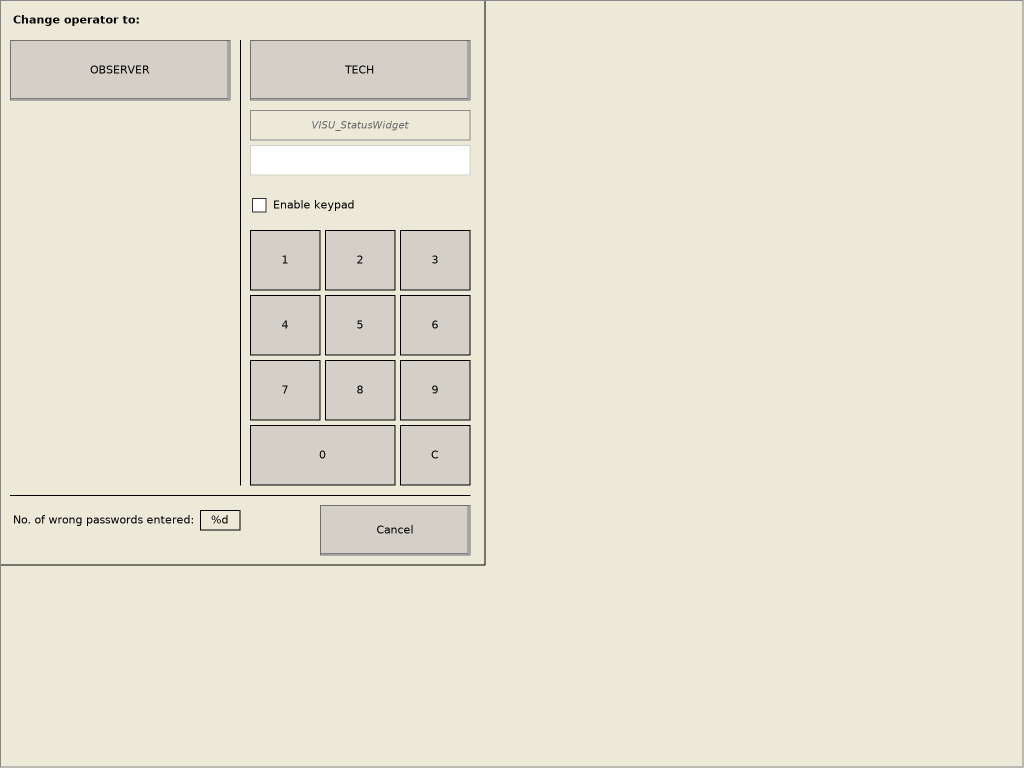
VISUALIZATION VISU_MTCSChangeOperatorDialog  // 1024x768
    Rectangle (0,0 485x565)
    Rectangle (250,230 70x60), "1", input disabled if: GLOBAL.gui.changeOperatorDialog.deactivate_keypad_keys
        OnMouseClick: execute { GLOBAL.gui.changeOperatorDialog.do_1 := TRUE; }
    Rectangle (325,230 70x60), "2", input disabled if: GLOBAL.gui.changeOperatorDialog.deactivate_keypad_keys
        OnMouseClick: execute { GLOBAL.gui.changeOperatorDialog.do_2 := TRUE; }
    Rectangle (400,230 70x60), "3", input disabled if: GLOBAL.gui.changeOperatorDialog.deactivate_keypad_keys
        OnMouseClick: execute { GLOBAL.gui.changeOperatorDialog.do_3 := TRUE; }
    Rectangle (250,295 70x60), "4", input disabled if: GLOBAL.gui.changeOperatorDialog.deactivate_keypad_keys
        OnMouseClick: execute { GLOBAL.gui.changeOperatorDialog.do_4 := TRUE; }
    Rectangle (325,295 70x60), "5", input disabled if: GLOBAL.gui.changeOperatorDialog.deactivate_keypad_keys
        OnMouseClick: execute { GLOBAL.gui.changeOperatorDialog.do_5 := TRUE; }
    Rectangle (400,295 70x60), "6", input disabled if: GLOBAL.gui.changeOperatorDialog.deactivate_keypad_keys
        OnMouseClick: execute { GLOBAL.gui.changeOperatorDialog.do_6 := TRUE; }
    Rectangle (250,360 70x60), "7", input disabled if: GLOBAL.gui.changeOperatorDialog.deactivate_keypad_keys
        OnMouseClick: execute { GLOBAL.gui.changeOperatorDialog.do_7 := TRUE; }
    Rectangle (325,360 70x60), "8", input disabled if: GLOBAL.gui.changeOperatorDialog.deactivate_keypad_keys
        OnMouseClick: execute { GLOBAL.gui.changeOperatorDialog.do_8 := TRUE; }
    Rectangle (400,360 70x60), "9", input disabled if: GLOBAL.gui.changeOperatorDialog.deactivate_keypad_keys
        OnMouseClick: execute { GLOBAL.gui.changeOperatorDialog.do_9 := TRUE; }
    Rectangle (250,425 145x60), "0", input disabled if: GLOBAL.gui.changeOperatorDialog.deactivate_keypad_keys
        OnMouseClick: execute { GLOBAL.gui.changeOperatorDialog.do_0 := TRUE; }
    Rectangle (400,425 70x60), "C", input disabled if: GLOBAL.gui.changeOperatorDialog.deactivate_keypad_keys
        OnMouseClick: execute { GLOBAL.gui.changeOperatorDialog.do_c := TRUE; }
    Button (320,505 150x50), "Cancel"
        OnMouseClick: execute { GLOBAL.gui.changeOperatorDialog.do_cancel := TRUE; }
        OnMouseClick: CloseDialog Dialog=VISU_MTCSChangeOperatorDialog, Result=Cancel, NumpadKeypadSet=True
    Line (10,495) (470,495)
    Label (10,10 120x20), "Change operator to:"
    Button (250,40 220x60), "TECH", input disabled if: GLOBAL.gui.changeOperatorDialog.deactivate_tech
        OnMouseClick: execute { GLOBAL.gui.changeOperatorDialog.do_tech := TRUE; }
        OnMouseClick: CloseDialog Dialog=VISU_MTCSChangeOperatorDialog, Result=OK, NumpadKeypadSet=True
    Button (10,40 220x60), "OBSERVER", input disabled if: GLOBAL.gui.changeOperatorDialog.deactivate_observer
        OnMouseClick: execute { GLOBAL.gui.changeOperatorDialog.do_observer := TRUE; }
        OnMouseClick: CloseDialog Dialog=VISU_MTCSChangeOperatorDialog, Result=OK, NumpadKeypadSet=True
    Line (240,40) (240,485)
    Frame (250,110 220x30)
        shows VISU_StatusWidget(widget := GLOBAL.gui.changeOperatorDialog.passwordHealthStatusWidget)
    Label (10,510 190x20), "No. of wrong passwords entered:"
    Rectangle (200,510 40x20), "%d", text variable: GLOBAL.mtcs.noOfFailedOperatorChanges
    Textfield (250,145 220x30), text variable: GLOBAL.gui.changeOperatorDialog._hiddenField, input disabled if: GLOBAL.gui.changeOperatorDialog.deactivate_keypad_checkbox
        OnMouseClick: write the text variable via Edit, password
    Checkbox (250,185 150x40), "Enable keypad", variable: GLOBAL.gui.changeOperatorDialog.keypadCheckbox, input disabled if: GLOBAL.gui.changeOperatorDialog.deactivate_keypad_checkbox
END_VISUALIZATION

(* stored: Version 1.1.0.1, ProductVersion 3.1.4019.2
   Visu VISU_MTCSChangeOperatorDialog: Id {f8de0c13-53e7-4026-8e75-c3e5e158ba8e} *)
